{attribute 'no_explicit_call' := 'do not call this function block directly'} 
FUNCTION_BLOCK OpcUaCommunicationSettings EXTENDS CommunicationSettings
VAR_INPUT
	ServerUrl : Tc2_System.T_MaxString;
	SessionConnectInfo : Tc3_PLCopen_OpcUa.ST_UASessionConnectInfo;
	ConnectionTimeout : TIME := Tc2_System.DEFAULT_ADS_TIMEOUT;
END_VAR
VAR
	_ClassName : STRING := __POUNAME();
END_VAR

PROPERTY CommunicationTypeName : STRING
GET
CommunicationTypeName := 'OPC-UA';
END_GET
END_PROPERTY

END_FUNCTION_BLOCK

(* stored: Version 1.1.0.1
   POU OpcUaCommunicationSettings: Id {c2bc7a85-877f-4176-b865-9a0e01611254}, SpecialFunc None
   Property CommunicationTypeName: Id {e2a50633-2698-4595-bba5-5e59f58f8df8}
   Get Get: Id {8a7a1051-aa7c-40be-8c59-31411120834e} *)
